{attribute addProperty BoxType "IODEVICETYPE_ETHERCATPROT"}
{attribute addProperty Id "Beckhoff_APS1xxxBeckhoff_APS1xxx_0455F8D34660582.5Beckhoff_APS4xxxBeckhoff_APS4xxx_87463DAF4804600.5SyncUnitsSyncUnits_CAB22D3B19524.375InputsInputs_C75D3FEC1280160OutputsOutputs_47D1E803848106InfoDataInfoData_E9F65A829612"}
{attribute addProperty CRC "1873596417"}
{attribute addProperty SizeInBites "11883"}
{attribute addProperty SizeInBytes "1485.375"}
TYPE EtherCAT_Master_APSxxxx_6FACD001 :
STRUCT
	{attribute addProperty Name "Beckhoff_APS1xxx"}
	Beckhoff_APS1xxx : Beckhoff_APS1xxx_0455F8D3;
	{attribute addProperty Name "Beckhoff_APS4xxx"}
	Beckhoff_APS4xxx : Beckhoff_APS4xxx_87463DAF;
	{attribute addProperty Name "SyncUnits"}
	SyncUnits : SyncUnits_CAB22D3B;
	{attribute addProperty Name "Inputs"}
	Inputs : Inputs_C75D3FEC;
	{attribute addProperty Name "Outputs"}
	Outputs : Outputs_47D1E803;
	{attribute addProperty Name "InfoData"}
	InfoData : InfoData_E9F65A82;
END_STRUCT
END_TYPE

(* stored: Version 1.2.0.0, ProductVersion 3.1.4024.9
   DUT EtherCAT_Master_APSxxxx_6FACD001: Id {73126df7-b94e-47dc-bfa4-18422113998c} *)
